Universal Robots PolyScope program: g_to_c.urp

Program g_to_c (installation=string_planes directory=/programs createdIn=5.17.3 lastSavedIn=5.17.3 robotSerialNumber=20245501435)
Calibrated DH parameters: a=[0.000154, -0.137004, -0.385524, -0.00002, 0.000092, 0]; d=[0.162441, 211.794786, -230.585024, 18.923638, 0.099786, 0.09951]; alpha=[1.569493, -0.001902, 0.003874, 1.570111, -1.570167, 0]; deltaTheta=[0, -1.242934, 1.056292, 0.186646, 0.000002, 0.000001]
InitVariablesNode
Robot Program (runOnlyOnce=false)
  MoveJ speed 60 deg/s, acceleration 80 deg/s^2 (useActiveTCP=true) feature=Base
    Waypoint Waypoint_1 (Relative): relativeFromPosition TCP in base x=267.761 y=455.827 z=63.349 mm, rx=-1.6064 ry=-1.9107 rz=0.8701 rad; joints [-141.614, -39.193, 108.912, -115.289, -70.779, -159.12] deg; TCP offset x=28.21 y=-96.107 z=-99.69 mm, rx=0 ry=0 rz=0 rad; TCP in base x=195.266 y=411.465 z=21.275 mm, rx=-1.7342 ry=-1.5169 rz=0.4321 rad; joints [-140.231, -30.937, 122.534, -154.989, -45.801, -143.196] deg
